// TwinCAT 3 PLC project PLC_v01
// ProgramVersion: 3.1.4022.1
// libraries:
//   Tc2_Math, * (Beckhoff Automation GmbH)
//   Tc2_MC2, * (Beckhoff Automation GmbH)
//   Tc2_MC2_Drive, * (Beckhoff Automation GmbH)
//   Tc2_NCI, * (Beckhoff Automation GmbH)
//   Tc2_NcKinematicTransformation, * (Beckhoff Automation GmbH)
//   Tc2_Standard, * (Beckhoff Automation GmbH)
//   Tc2_System, * (Beckhoff Automation GmbH)
//   Tc2_Utilities, * (Beckhoff Automation GmbH)
//   Tc3_Module, * (Beckhoff Automation GmbH)
//   Tc3_PLCopen_OpcUa, * (Beckhoff Automation GmbH)
//   VisuDialogs, * (System)
// project tree:
//   DUTs/ E_NciChannelState.TcDUT, ST_AxisInterface.TcDUT, ST_AxisInterfaceIn.TcDUT, ST_AxisInterfaceOut.TcDUT, ST_FileDialogParams.TcDUT, ST_OpcUAVariablesR.TcDUT, ST_OpcUAVariablesW.TcDUT (not stored)
//   GVLs/ GVL_Axis.TcGVL, GVL_FileOpen.TcGVL (not stored), GVL_Kin.TcGVL, GVL_Nci.TcGVL, GVL_Process.TcGVL (not stored), GVL_Process_Deneme.TcGVL
//   / PlcTask.TcTTO, Visualization Manager.TcVMO (not stored)
//   POUs/Deneme/ POU_Process_Deneme.TcPOU, POU_VisButton.TcPOU
//   POUs/ FB_AxisControl.TcPOU (not stored), MAIN.TcPOU, PRG_MFuncControl.TcPOU (not stored), PRG_NcControl.TcPOU, PRG_Process.TcPOU (not stored)
//   POUs/KIN/ PRG_Kinematic.TcPOU
//   POUs/NCI/ FB_NciChannel.TcPOU (not stored), FB_NciFastMFunctions.TcPOU, FB_NciMFunctions.TcPOU (not stored), FB_NciReadLine.TcPOU (not stored), FB_NciWriteToolParams.TcPOU (not stored)
//   POUs/OPC-UA/ FB_OpcUAWrite.TcPOU (not stored), PRG_OpcUA.TcPOU (not stored)
//   POUs/UTIL/ FB_Flash.TcPOU (not stored), FB_ScreenOnOff_Win7.TcPOU
//   VISUs/AxisList/ VisuAxisM1.TcVIS, VisuAxisM2.TcVIS, VisuAxisM3.TcVIS, VisuAxisX.TcVIS (not stored), VisuAxisX_1.TcVIS, VisuAxisY.TcVIS, VisuAxisY_1.TcVIS, VisuAxisZ.TcVIS (not stored), VisuAxisZ_1.TcVIS (not stored)
//   VISUs/Frame/ Visualization_FileList.TcVIS, VisuAxisControl.TcVIS, VisuAxisControl_1.TcVIS, VisuAxisInfo.TcVIS (not stored)
//   VISUs/ GlobalTextList.TcGTLO, ImagePool.TcIPO (not stored), Visualization.TcVIS (not stored), Visualization_1.TcVIS, Visualization_AxesInfo.TcVIS, Visualization_AxesInfo_Manual.TcVIS
// real-time tasks:
//   TASK PlcTask: cycle T#10ms, priority 20, ADS port 350
// motion (NC):
//   TASK NC-Task 1 SAF: cycle T#2ms, priority 4, ADS port 501
//   TASK NC-Task 1 SVB: cycle T#10ms, priority 8, ADS port 511
//   AXIS M1 (id 1)
//     Dynamic: Acceleration=120.484, Deceleration=120.484, Jerk=361.452, DelayTime=0.008
//     Velo: RefSearch=0.803225806425292, RefSync=0.803225806425292, SlowManual=10, FastManual=25, Fast=80.3225806425291, Maximum=80.3226
//     OtherSettings: AllowMotionCmdToSlave=true
//     encoder EncType=1
//       EncPara: ScaleFactorNumerator=11.6129032254259, ScaleFactorDenominator=1048576, Offset=-0.7867, Inverse=true
//     drive DrvType=5
//       DrvPara: Inverse=true
//         Analog: VeloReferenz=88.3548387067821, TorqueScale=10, ScaleFactorActTorque=0.1
//         TimeComp: TaskDelayCycles=1
//     controller CtrType=1
//       CtrPara: PriorControlFactor=1
//         PID: PosKp=10
//         Observer: BandWidth=20
//   AXIS M2 (id 2)
//     Dynamic: Acceleration=120.483870963794, Deceleration=120.483870963794, Jerk=361.451612891381, DelayTime=0.008
//     Velo: RefSearch=0.803225806425292, RefSync=0.803225806425292, SlowManual=10, FastManual=25, Fast=80.3225806425291, Maximum=80.3225806425291
//     OtherSettings: AllowMotionCmdToSlave=true
//     encoder EncType=1
//       EncPara: ScaleFactorNumerator=11.6129032254259, ScaleFactorDenominator=1048576, Offset=-4.6881, Inverse=true
//     drive DrvType=5
//       DrvPara: Inverse=true
//         Analog: VeloReferenz=88.3548387067821, TorqueScale=10, ScaleFactorActTorque=0.1
//         TimeComp: TaskDelayCycles=1
//     controller CtrType=1
//       CtrPara: PriorControlFactor=1
//         PID: PosKp=10
//         Observer: BandWidth=20
//   AXIS M3 (id 3)
//     Dynamic: Acceleration=120.483870963794, Deceleration=120.483870963794, Jerk=361.451612891381, DelayTime=0.008
//     Velo: RefSearch=0.803225806425292, RefSync=0.803225806425292, SlowManual=10, FastManual=25, Fast=80.3225806425291, Maximum=80.3225806425291
//     OtherSettings: AllowMotionCmdToSlave=true
//     encoder EncType=1
//       EncPara: ScaleFactorNumerator=11.6129032254259, ScaleFactorDenominator=1048576, Offset=4810.3626, Inverse=true
//     drive DrvType=5
//       DrvPara: Inverse=true
//         Analog: VeloReferenz=88.3548387067821, TorqueScale=10, ScaleFactorActTorque=0.1
//         TimeComp: TaskDelayCycles=1
//     controller CtrType=1
//       CtrPara: PriorControlFactor=1
//         PID: PosKp=10
//         Observer: BandWidth=20
//   AXIS X (id 4)
//     OtherSettings: AllowMotionCmdToSlave=true
//     encoder EncType=1
//     drive DrvType=5
//       Analog: ScaleFactorActTorque=0.1
//       TimeComp: TaskDelayCycles=1
//     controller CtrType=1
//       CtrPara: PriorControlFactor=1
//         Observer: BandWidth=20
//   AXIS Y (id 5)
//     OtherSettings: AllowMotionCmdToSlave=true
//     encoder EncType=1
//     drive DrvType=5
//       Analog: ScaleFactorActTorque=0.1
//       TimeComp: TaskDelayCycles=1
//     controller CtrType=1
//       CtrPara: PriorControlFactor=1
//         Observer: BandWidth=20
//   AXIS Z (id 6)
//     OtherSettings: AllowMotionCmdToSlave=true
//     encoder EncType=1
//     drive DrvType=5
//       Analog: ScaleFactorActTorque=0.1
//       TimeComp: TaskDelayCycles=1
//     controller CtrType=1
//       CtrPara: PriorControlFactor=1
//         Observer: BandWidth=20
// I/O:
//   DEVICE Device 1 (EtherCAT) (disabled), AmsNetId 10.70.16.23.2.1
//     Term 1 (EK1200) [EK1200-5000 EtherCAT Power supply (2A E-Bus)]
//       Term 2 (EL1008) [EL1008 8Ch. Dig. Input 24V, 3ms]
//       Term 3 (EL2008) [EL2008 8Ch. Dig. Output 24V, 0.5A]
//       Term 4 (EL9576) [EL9576 Brake chopper terminal]
//       Term 5 (EL7211-0010) [EL7211-0010 1Ch. MDP742 Servo motor output stage with OCT (50V, 4.5A RMS)]
//       Term 6 (EL7211-0010) [EL7211-0010 1Ch. MDP742 Servo motor output stage with OCT (50V, 4.5A RMS)]
//       Term 7 (EL7211-0010) [EL7211-0010 1Ch. MDP742 Servo motor output stage with OCT (50V, 4.5A RMS)]
//       Term 8 (EL9011) [EL9011 End Terminal]
// variable links:
//   PLC_v01/PLC_v01 Instance <-> NC-Task 1 SAF/Axes/M1
//     PlcTask Inputs/GVL_Axis.AxisM1_B.NcToPlc <-> Outputs/ToPlc
//     PlcTask Outputs/GVL_Axis.AxisM1_B.PlcToNc <-> Inputs/FromPlc
//   PLC_v01/PLC_v01 Instance <-> NC-Task 1 SAF/Axes/M2
//     PlcTask Inputs/GVL_Axis.AxisM2_C.NcToPlc <-> Outputs/ToPlc
//     PlcTask Outputs/GVL_Axis.AxisM2_C.PlcToNc <-> Inputs/FromPlc
//   PLC_v01/PLC_v01 Instance <-> NC-Task 1 SAF/Axes/M3
//     PlcTask Inputs/GVL_Axis.AxisM3_A.NcToPlc <-> Outputs/ToPlc
//     PlcTask Outputs/GVL_Axis.AxisM3_A.PlcToNc <-> Inputs/FromPlc
//   PLC_v01/PLC_v01 Instance <-> NC-Task 1 SAF/Axes/X
//     PlcTask Inputs/GVL_Axis.AxisX.NcToPlc <-> Outputs/ToPlc
//     PlcTask Outputs/GVL_Axis.AxisX.PlcToNc <-> Inputs/FromPlc
//   PLC_v01/PLC_v01 Instance <-> NC-Task 1 SAF/Axes/Y
//     PlcTask Inputs/GVL_Axis.AxisY.NcToPlc <-> Outputs/ToPlc
//     PlcTask Outputs/GVL_Axis.AxisY.PlcToNc <-> Inputs/FromPlc
//   PLC_v01/PLC_v01 Instance <-> NC-Task 1 SAF/Axes/Z
//     PlcTask Inputs/GVL_Axis.AxisZ.NcToPlc <-> Outputs/ToPlc
//     PlcTask Outputs/GVL_Axis.AxisZ.PlcToNc <-> Inputs/FromPlc
//   PLC_v01/PLC_v01 Instance <-> NC-Task 1 SAF/KIN
//     PlcTask Inputs/GVL_Kin.stKinToPLC <-> Outputs/ToPlc
//     PlcTask Outputs/GVL_Kin.stKinFromPLC <-> Inputs/FromPlc
//   PLC_v01/PLC_v01 Instance <-> NC-Task 1 SAF/NCI
//     PlcTask Inputs/GVL_Nci.stNciToPLC <-> Outputs/ToPlc
//     PlcTask Outputs/GVL_Nci.stPlcToNci <-> Inputs/FromPlc

CONFIGURATION PLC_v01
    RESOURCE PLC ON TwinCAT3
        TASK PlcTask(INTERVAL := T#10ms, PRIORITY := 20);
        PROGRAM MAIN WITH PlcTask : MAIN;
    END_RESOURCE
END_CONFIGURATION

// ---- DUTs/E_NciChannelState.TcDUT
TYPE E_NciChannelState :
(
	eNCI_INTERPRETER_INITFAILED := 0, 
	eNCI_INTERPRETER_IDLE := 1, 
	eNCI_INTERPRETER_READY := 2,
	eNCI_INTERPRETER_STARTED := 3, 
	eNCI_INTERPRETER_SCANNING := 4, 
	eNCI_INTERPRETER_RUNNING := 5,
	eNCI_INTERPRETER_STAY_RUNNING := 6,
	eNCI_INTERPRETER_WRITETABLE := 7,
	eNCI_INTERPRETER_SEARCHLINE := 8, 
	eNCI_INTERPRETER_END := 9,
	eNCI_INTERPRETER_SINGLESTOP := 10,
	eNCI_INTERPRETER_ABORTING := 11,
	eNCI_INTERPRETER_ABORTED := 12, 
	eNCI_INTERPRETER_FAULT := 13,
	eNCI_INTERPRETER_RESET := 14, 
	eNCI_INTERPRETER_STOP := 15,
	eNCI_INTERPRETER_WAITFUNC := 16,
	eNCI_INTERPRETER_FLUSHBUFFERS := 17
);
END_TYPE

// ---- DUTs/ST_AxisInterface.TcDUT
TYPE ST_AxisInterface :
STRUCT
	In		: ST_AxisInterfaceIn;
	Out		: ST_AxisInterfaceOut;
END_STRUCT
END_TYPE

// ---- DUTs/ST_AxisInterfaceIn.TcDUT
TYPE ST_AxisInterfaceIn :
STRUCT
	xEnable			: BOOL;
	xReset			: BOOL;
	xDriveReset		: BOOL;
	xMove			: BOOL;
	xHome			: BOOL;
	xHomeSensor		: BOOL;
	xJogFw			: BOOL;
	xJogBw			: BOOL;
	fHomePos		: LREAL;
	fSetPos			: LREAL;
	fSetVelo		: LREAL;
	fSetAcc			: LREAL;
	fSetDec			: LREAL;
	fSetJerk		: LREAL;
	fJogVelo		: LREAL	:= 20;
	fOverride		: LREAL	:= 100.0;
END_STRUCT
END_TYPE

// ---- DUTs/ST_AxisInterfaceOut.TcDUT
TYPE ST_AxisInterfaceOut :
STRUCT
	xEnabled		: BOOL;
	xHomed			: BOOL;
	xMoveDone		: BOOL;
	xAxisError		: BOOL;
	nAxisErrId		: UDINT;
	xDriveError		: BOOL;
	nDriveErrId		: UDINT;
	xFunctionError	: BOOL;
	nFunctionErrId	: UDINT;
END_STRUCT
END_TYPE

// ---- DUTs/ST_FileDialogParams.TcDUT
TYPE ST_FileDialogParams :
STRUCT
	sTitle 		: STRING;
	sDirectory 	: STRING(255);
	sFile 		: STRING(255);
	sFilter 	: STRING;
	bInit 		: BOOL;
END_STRUCT
END_TYPE

// ---- DUTs/ST_OpcUAVariablesR.TcDUT
TYPE ST_OpcUAVariablesR :
STRUCT
	bEnableAllProcess	: BOOL;
	bNciStart			: BOOL;
END_STRUCT
END_TYPE

// ---- GVLs/GVL_Axis.TcGVL
VAR_GLOBAL
// Kullanilacak olan gercek eksenler
	AxisM1_B			: AXIS_REF;			
	AxisM2_C			: AXIS_REF;
	AxisM3_A			: AXIS_REF;	
	
// Kinematik grupta olusacak eksenler
	AxisX				: AXIS_REF;
	AxisY				: AXIS_REF;
	AxisZ				: AXIS_REF;
	
// Gercek eksenler icin interface yapilari
	stAxisM1_B			: ST_AxisInterface;
	stAxisM2_C			: ST_AxisInterface;
	stAxisM3_A			: ST_AxisInterface;
	
// Kinematik eksenlerin interface yapilari
	stAxisX				: ST_AxisInterface;
	stAxisY				: ST_AxisInterface;
	stAxisZ				: ST_AxisInterface;
	
	sAxisM1_BName		: STRING	:= 'Axis M1';
	sAxisM2_CName		: STRING	:= 'Axis M2';
	sAxisM3_AName		: STRING	:= 'Axis M3';
	
	
	sAxisXName			: STRING	:= 'Axis X';
	sAxisYName			: STRING	:= 'Axis Y';
	sAxisZName			: STRING	:= 'Axis Z';
	
	AxisM1PosValue		: LREAL;
	AxisM2PosValue		: LREAL;
	AxisM3PosValue		: LREAL;
	
	AxisXVal	:	LREAL;
	AxisYVal	:	LREAL;	
	AxisZVal	:	LREAL;
	
END_VAR

// ---- GVLs/GVL_Kin.TcGVL
{attribute 'qualified_only'}
VAR_GLOBAL
	stKinToPLC			AT%I*	: NCTOPLC_NCICHANNEL_REF;
	stKinFromPLC		AT%Q*	: PLCTONC_NCICHANNEL_REF;
	
	stAxesList					: ST_KinAxes;
	
END_VAR

// ---- GVLs/GVL_Nci.TcGVL
VAR_GLOBAL
	stNciToPLC	AT%I*		: NCTOPLC_NCICHANNEL_REF;
	stPlcToNci	AT%Q*		: PLCTONC_NCICHANNEL_REF;
	
	bMFunc					: ARRAY[0..cnMaxMFuncNumber] OF BOOL;
	bQuitMFunc				: ARRAY[0..cnMaxMFuncNumber] OF BOOL;
	bFastMFunc				: ARRAY[0..cnMaxMFuncNumber] OF BOOL;
	
	fNciRParamsWrite		: ARRAY[cnStartIndexWriteRParam..cnEndIndexWriteRParam] OF LREAL;
	fNciRParamsRead			: ARRAY[cnStartIndexReadRParam..cnEndIndexReadRParam] OF LREAL;
	stNciToolParams			: ARRAY[1..cnMaxToolNumber] OF ToolDesc;
END_VAR
VAR_GLOBAL CONSTANT
	cnMaxMFuncNumber		: INT	:= 159;
	cnStartIndexWriteRParam	: INT	:= 0;
	cnEndIndexWriteRParam	: INT	:= 100;
	cnStartIndexReadRParam	: INT	:= 101;
	cnEndIndexReadRParam	: INT	:= 201;
	cnMaxToolNumber			: INT	:= 10;
END_VAR

// ---- GVLs/GVL_Process_Deneme.TcGVL
{attribute 'qualified_only'}
VAR_GLOBAL
	
bSensor	:	BOOL;
bCatch	:	BOOL;

bMovementDone	:	BOOL;
bDataComp	:	BOOL;
bGrapDone	:	BOOL;
END_VAR

// ---- POUs/MAIN.TcPOU
PROGRAM MAIN
VAR
	sFilePathName	: STRING := 'C:\TwinCAT\CNC\TestNci1.txt';
	sErrorMessage	: STRING := '';
	bOpen			: BOOL;
	bClose 			: BOOL;
	bSave 			: BOOL;
	bNew			: BOOL;
	nErrorCode		: USINT;
	nLineNumber		: USINT;
	bEnable: BOOL;
END_VAR



sErrorMessage	:= VisuFctTextEditorGetErrorText(usiErrCode := nErrorCode);

PRG_NcControl();
//PRG_MFuncControl();
PRG_Kinematic();

//PRG_Process();

//PRG_OpcUA();

//POU_VisButton();
POU_Process_Deneme();


	PRG_Kinematic.bExecuteKinConfigGroup;
	
	
	stAxisX.In.fSetPos;
	stAxisY.In.fSetPos;
	stAxisZ.In.fSetPos;

	
	stAxisX.In.xMove;
	stAxisY.In.xMove;
	stAxisZ.In.xMove;



AxisM1PosValue	:=	LMOD(AxisM1_B.NcToPlc.ModuloActPos,360);
AxisM2PosValue	:=	LMOD(AxisM2_C.NcToPlc.ModuloActPos,360);
AxisM3PosValue	:=	LMOD(AxisM3_A.NcToPlc.ModuloActPos,360);



	
	
	AxisXVal	:=	AxisX.NcToPlc.ActPos;
	AxisYVal	:=	AxisY.NcToPlc.ActPos;
	AxisZVal	:=	AxisZ.NcToPlc.ActPos;

END_PROGRAM

// ---- POUs/PRG_NcControl.TcPOU
PROGRAM PRG_NcControl
VAR_INPUT
	//PRG_Process içerisinde resetlemede kullanabilmek için 
	bNciEnable			: BOOL;
	bNciStart			: BOOL;
END_VAR

VAR
	fbAxisControlM1_B	: FB_AxisControl;
	fbAxisControlM2_C	: FB_AxisControl;
	fbAxisControlM3_A	: FB_AxisControl;	
	
	fbAxisControlX		: FB_AxisControl;
	fbAxisControlY		: FB_AxisControl;
	fbAxisControlZ		: FB_AxisControl;
	
	fbNciChannel		: FB_NciChannel;
	fbNciMFunc			: FB_NciMFunctions;
	fbNciFastMFunc		: FB_NciFastMFunctions;
	fbNciReadLine		: FB_NciReadLine;
	bAxisEnable			: BOOL;
	fAxisOverride		: LREAL;
	bNciSingleMode		: BOOL;
	bNciNextStep		: BOOL;
	fNciOverride		: LREAL	:= 100.0;
	eNciItpState		: E_NciChannelState;
	bBuildGroupDone		: BOOL;
	bSingleModeActive	: BOOL;
	bProgramRunning		: BOOL;
	bProgramStopped		: BOOL;
	bProgramFinished	: BOOL;
	bNciError			: BOOL;
	nNciErrorId			: UDINT;
	bMFuncBusy			: BOOL;
	bMFuncError			: BOOL;
	nMFuncErrorId		: UDINT;
	bEnableReadLine		: BOOL	:= TRUE;
	sNciLines			: STRING(255);
	sNciActualLine		: STRING(80);	
	bEnable: BOOL;
END_VAR

//ACT_EmergencyOnPanel();

fbAxisControlM1_B(stAxisInterface:= stAxisM1_B, stAxisRef:= AxisM1_B);
fbAxisControlM2_C(stAxisInterface:= stAxisM2_C, stAxisRef:= AxisM2_C);
fbAxisControlM3_A(stAxisInterface:= stAxisM3_A, stAxisRef:= AxisM3_A);

fbAxisControlX(stAxisInterface:= stAxisX, stAxisRef:= AxisX);
fbAxisControlY(stAxisInterface:= stAxisY, stAxisRef:= AxisY);
fbAxisControlZ(stAxisInterface:= stAxisZ, stAxisRef:= AxisZ);

(*
		stAxisX.In.xEnable		:= bEnable;
		stAxisY.In.xEnable		:= bEnable;
		stAxisZ.In.xEnable		:= bEnable;
		stAxisM1_B.In.xEnable	:= bEnable;
		stAxisM2_C.In.xEnable	:= bEnable;
		stAxisM3_A.In.xEnable	:= bEnable;
*)
(*		
fbNciChannel(
	bEnable				:= bNciEnable, 
	bStart				:= bNciStart, 
	bSingleMode			:= bNciSingleMode,
	bSingleModeStart	:= bNciNextStep,
	fOverride			:= fNciOverride,
	nXAxisId			:= AxisX.NcToPlc.AxisId, 
	nYAxisId			:= AxisY.NcToPlc.AxisId, 
	nZAxisId			:= AxisZ.NcToPlc.AxisId, 
	sProgramPath		:= PRG_Process.sFileName, 
	sSubroutinePath		:= 'C:\TwinCAT\Mc\Nci\Sub\', 
	sNciToPLC			:= stNciToPLC, 
	sPlcToNci			:= stPlcToNci, 
	eNciChannelState	=> eNciItpState, 
	bBuildGroupDone		=> bBuildGroupDone, 
	bSingleModeActive	=> bSingleModeActive,
	bProgramRunning		=> bProgramRunning, 
	bProgramStopped		=> bProgramStopped, 
	bProgramFinished	=> bProgramFinished, 
	bError				=> bNciError, 
	nErrorId			=> nNciErrorId);
	
fbNciMFunc(
	sNciToPlc			:= stNciToPLC, 
	sPlcToNci			:= stPlcToNci, 
	bBusy				=> bMFuncBusy, 
	bError				=> bMFuncError, 
	nErrorId			=> nMFuncErrorId);
	
fbNciFastMFunc(
	sNciToPlc			:= stNciToPLC);
	
fbNciReadLine(
	bEnable				:= bEnableReadLine, 
	tIdleTime			:= T#100MS, 
	sNciToPlc			:= stNciToPLC, 
	sNciLines			=> sNciLines,
	sActualLine			=> sNciActualLine );
	

*)

ACTION ACT_EmergencyOnPanel:
(*Button On Control Panel- Emergency and Green Button*)
GVL_Process.fTrigbEmergency(CLK:= GVL_Process.bEmergencyOnPanel);
GVL_Process.rTrigbEmergency(CLK:= GVL_Process.bEmergencyOnPanel);


CASE GVL_Process.nStateEmergency OF 
0:
	IF GVL_Process.fTrigbEmergency.Q THEN 
		fNciOverride	:= 0;
		GVL_Process.nStateEmergency	:= 10;
	END_IF
	
10:
	IF GVL_Process.rTrigbEmergency.Q THEN 
		GVL_Process.nStateEmergency	:= 20;
	END_IF
	
20:
	IF GVL_Process.bGreenBtnOnPanel THEN 
		fNciOverride	:= 100;
		GVL_Process.nStateEmergency	:= 0;
	END_IF
END_CASE
END_ACTION

END_PROGRAM

// ---- POUs/NCI/FB_NciFastMFunctions.TcPOU
FUNCTION_BLOCK FB_NciFastMFunctions
VAR_IN_OUT
	sNciToPlc		: NCTOPLC_NCICHANNEL_REF;
END_VAR
VAR_OUTPUT
END_VAR
VAR
	i				: INT;
	l				: SINT;
	bBit			: BOOL;
	index			: UINT;
END_VAR


(* Fill the global defined M-functions array with 
	fast M-Functions from NCI Channel *)

FOR i:=0 TO 4 DO  (* check all 5 dwords *)
	FOR l := 0 TO 31 DO
		bBit := GETBIT32(sNciToPlc.FastMFuncMask[i+1], l);
      	index := INT_TO_UINT((i*32) + l);
		IF ( bBit ) THEN
			bFastMFunc[index] := TRUE;
		ELSE
			bFastMFunc[index] := FALSE;
		END_IF
	END_FOR
END_FOR

END_FUNCTION_BLOCK

// ---- POUs/KIN/PRG_Kinematic.TcPOU
PROGRAM PRG_Kinematic
VAR_INPUT
		bExecuteKinConfigGroup	: BOOL;
		bCartesianMode			: BOOL := TRUE;
		bExecuteKinResetGroup	: BOOL;
END_VAR
VAR
	fbKinConfigGroup			: FB_KinConfigGroup;
	fbKinResetGroup				: FB_KinResetGroup;
	eKinStatus					: E_KinStatus;
END_VAR


GVL_Kin.stAxesList.nAxisIdsAcs[1]	:= AxisM1_B.NcToPlc.AxisId;
GVL_Kin.stAxesList.nAxisIdsAcs[2]	:= AxisM2_C.NcToPlc.AxisId;
GVL_Kin.stAxesList.nAxisIdsAcs[3]	:= AxisM3_A.NcToPlc.AxisId;

GVL_Kin.stAxesList.nAxisIdsMcs[1]	:= AxisX.NcToPlc.AxisId;
GVL_Kin.stAxesList.nAxisIdsMcs[2]	:= AxisY.NcToPlc.AxisId;
GVL_Kin.stAxesList.nAxisIdsMcs[3]	:= AxisZ.NcToPlc.AxisId;

ItpSetOverridePercent(100.0, GVL_Kin.stKinFromPLC);

fbKinConfigGroup(
	bExecute		:= bExecuteKinConfigGroup, 
	bCartesianMode	:= bCartesianMode, 
	stAxesList		:= GVL_Kin.stAxesList, 
	stKinRefIn		:= GVL_Kin.stKinToPLC);	
	
fbKinResetGroup(
	bExecute		:= bExecuteKinResetGroup, 
	nItpChannelId	:= ItpGetChannelId(GVL_Kin.stKinToPLC), 
	stKinRefIn		:= GVL_Kin.stKinToPLC, 
	stAxesList		:= GVL_Kin.stAxesList);

END_PROGRAM

// ---- POUs/Deneme/POU_Process_Deneme.TcPOU
PROGRAM POU_Process_Deneme
VAR
	nStateProcess: INT;
	bSystemStart: BOOL;
	bSensor: BOOL;
	T1: TON;
	T2: TON;
	rtrig_Obj: R_TRIG;
END_VAR

		
	stAxisM1_B.In.xEnable	:= TRUE;
	stAxisM2_C.In.xEnable	:= TRUE;
	stAxisM3_A.In.xEnable	:= TRUE;
	
	stAxisX.In.xEnable	:= TRUE;
	stAxisY.In.xEnable	:= TRUE;
	stAxisZ.In.xEnable	:= TRUE;
		
	stAxisM1_B.In.fOverride	:= 100;
	stAxisM2_C.In.fOverride	:= 100;
	stAxisM3_A.In.fOverride	:= 100;
	
	stAxisX.In.fOverride	:= 100;
	stAxisY.In.fOverride	:= 100;
	stAxisZ.In.fOverride	:= 100;
	

	
CASE nStateProcess	OF
	
0:
IF bSystemStart THEN


	PRG_Kinematic.bExecuteKinConfigGroup	:=	TRUE;
	stAxisX.In.xMove	:=	TRUE;
	stAxisY.In.xMove	:=	TRUE;
	stAxisZ.In.xMove	:=	TRUE;

			
	stAxisX.In.fSetVelo	:=50;
	stAxisY.In.fSetVelo	:=50;
	stAxisZ.In.fSetVelo	:=50;

	IF 
	PRG_Kinematic.fbKinConfigGroup.bDone AND 
	stAxisX.Out.xEnabled	AND
	stAxisY.Out.xEnabled	AND
	stAxisZ.Out.xEnabled	THEN
	
	

		nStateProcess	:=	10;
	
	ELSIF	PRG_Kinematic.fbKinConfigGroup.bError THEN
		nStateProcess	:=	1000;
	END_IF	
	
END_IF

10:
GVL_Process_Deneme.bMovementDone	:=	FALSE;
GVL_Process_Deneme.bDataComp	:=FALSE;


IF	GVL_Process_Deneme.bSensor	THEN
	
	GVL_Process_Deneme.bMovementDone	:=	TRUE;
	
	stAxisX.In.fSetPos	:=	0;
	stAxisY.In.fSetPos	:=	0;
	stAxisZ.In.fSetPos	:=	-400;
	

	IF 	stAxisX.Out.xMoveDone	AND stAxisY.Out.xMoveDone	AND stAxisZ.Out.xMoveDone THEN 
	
	GVL_Process_Deneme.bCatch	:=	TRUE;
	
	GVL_Process_Deneme.bMovementDone	:=	FALSE;				//Malzeme Alındı


	
	nStateProcess	:=	20;
	
	ELSIF stAxisX.Out.xAxisError	OR
	stAxisY.Out.xAxisError	OR
	stAxisZ.Out.xAxisError	OR
	stAxisM1_B.Out.xAxisError	OR
	stAxisM2_C.Out.xAxisError	OR	
	stAxisM3_A.Out.xAxisError	THEN

	nStateProcess	:=	999;	
	
END_IF
	
	
	
END_IF

20:

stAxisX.In.fSetVelo	:=300;
stAxisY.In.fSetVelo	:=300;
stAxisZ.In.fSetVelo	:=300;


stAxisZ.In.fSetPos	:=	-370;			//Alınan malzeme bırakılacağı konuma götürüldü
stAxisY.In.fSetPos	:=	310;

nStateProcess	:=	25;


25:

	IF  stAxisY.Out.xMoveDone	AND stAxisZ.Out.xMoveDone THEN 

	
	nStateProcess	:=	30;
	
	ELSIF stAxisX.Out.xAxisError	OR
	stAxisY.Out.xAxisError	OR
	stAxisZ.Out.xAxisError	OR
	stAxisM1_B.Out.xAxisError	OR
	stAxisM2_C.Out.xAxisError	OR	
	stAxisM3_A.Out.xAxisError	THEN

	nStateProcess	:=	999;	
	
END_IF
	
30:
stAxisX.In.fSetVelo	:=50;
stAxisY.In.fSetVelo	:=50;
stAxisZ.In.fSetVelo	:=50;

stAxisZ.In.fSetPos	:=	-400;		



	IF stAxisZ.Out.xMoveDone THEN 

	GVL_Process_Deneme.bDataComp	:=	TRUE;	// Malzeme bırakıldı
	
//	GVL_Process_Deneme.bMovementDone	:=	TRUE;

	GVL_Process_Deneme.bCatch	:=	FALSE;
	
	
	nStateProcess	:=	40;
	
	
	ELSIF stAxisX.Out.xAxisError	OR
	stAxisY.Out.xAxisError	OR
	stAxisZ.Out.xAxisError	OR
	stAxisM1_B.Out.xAxisError	OR
	stAxisM2_C.Out.xAxisError	OR	
	stAxisM3_A.Out.xAxisError	THEN

	nStateProcess	:=	999;	
	
END_IF


40:

stAxisX.In.fSetVelo	:=1000;
stAxisY.In.fSetVelo	:=1000;
stAxisZ.In.fSetVelo	:=1000;


stAxisX.In.fSetPos	:=	0;
stAxisY.In.fSetPos	:=	0;
stAxisZ.In.fSetPos	:=	-370;

nStateProcess	:=	45;

45:
		
	IF 	stAxisX.Out.xMoveDone	AND stAxisY.Out.xMoveDone	 THEN 


	GVL_Process_Deneme.bDataComp	:=FALSE;
		GVL_Process_Deneme.bMovementDone	:=FALSE;

	
	nStateProcess	:=	0;
	
	
	ELSIF stAxisX.Out.xAxisError	OR
	stAxisY.Out.xAxisError	OR
	stAxisZ.Out.xAxisError	OR
	stAxisM1_B.Out.xAxisError	OR
	stAxisM2_C.Out.xAxisError	OR	
	stAxisM3_A.Out.xAxisError	THEN

	nStateProcess	:=	999;	
	
END_IF





END_CASE

END_PROGRAM

// ---- POUs/Deneme/POU_VisButton.TcPOU
PROGRAM POU_VisButton
VAR
	
xUp	:	BOOL;
xDown	:	BOOL;

yUp	:	BOOL;
yDown	:	BOOL;

zuP	:	BOOL;	
zDown	:	BOOL;

DecVal	:	LREAL;



	xUpR_TRIG: R_TRIG;
	xDownR_TRIG: R_TRIG;
	yUpR_TRIG: R_TRIG;
	yDownR_TRIG: R_TRIG;
	zUpR_TRIG: R_TRIG;
	zDownR_TRIG: R_TRIG;
	BridgeValZ: LREAL;
END_VAR

	
xUpR_TRIG(CLK:=xUp , Q=> );
xDownR_TRIG(CLK:=xDown , Q=> );

yUpR_TRIG(CLK:=yUp , Q=> );
yDownR_TRIG(CLK:=yDown , Q=> );

zUpR_TRIG(CLK:=zUp , Q=> );
zDownR_TRIG(CLK:=zDown , Q=> );


stAxisZ.In.fSetPos	:=	BridgeValZ;

	//stAxisX.In.fSetPos;
	//stAxisY.In.fSetPos;
	//stAxisZ.In.fSetPos;

IF xUpR_TRIG.Q	THEN
	
stAxisX.In.fSetPos	:=	stAxisX.In.fSetPos	+	10;


ELSIF xDownR_TRIG.Q THEN
	stAxisX.In.fSetPos	:=	stAxisX.In.fSetPos	-	10;
END_IF



IF yUpR_TRIG.Q	THEN
	
stAxisY.In.fSetPos	:=	stAxisY.In.fSetPos	+	10;


ELSIF yDownR_TRIG.Q THEN
	stAxisY.In.fSetPos	:=	stAxisY.In.fSetPos	-	10;
END_IF




IF zUpR_TRIG.Q	THEN
	
BridgeValZ	:=	BridgeValZ	+	10;


ELSIF zDownR_TRIG.Q THEN
	BridgeValZ	:=	BridgeValZ	-	10;
END_IF

END_PROGRAM

// ---- POUs/UTIL/FB_ScreenOnOff_Win7.TcPOU
FUNCTION_BLOCK FB_ScreenOnOff_Win7
VAR_INPUT
	bScreenOff			: BOOL;
END_VAR
VAR_OUTPUT
	bDone				: BOOL;
END_VAR
VAR
	fbSleepMonitor		: NT_StartProcess;
	nState				: INT;
END_VAR

CASE nState OF 	
0:
	IF bScreenOff THEN
		nState	:= 10;
	END_IF
	
10:
	fbSleepMonitor(
		NETID		:= '', 
		PATHSTR		:= 'C:\MonitorSleep.exe', 
		DIRNAME		:= 'C:\', 
		COMNDLINE	:= , 
		START		:= TRUE, 
		TMOUT		:= T#5S, 
		BUSY		=> , 
		ERR			=> , 
		ERRID		=> );
	
	IF NOT fbSleepMonitor.BUSY AND NOT fbSleepMonitor.ERR THEN 
		fbSleepMonitor(START := FALSE);
		nState		:= 20;
	END_IF 
		
20:
	bDone	:= TRUE;
	IF NOT bScreenOff THEN 
		bDone 	:= FALSE;
		nState	:= 0;
	END_IF 		

END_CASE

END_FUNCTION_BLOCK

// ---- VISUs/AxisList/VisuAxisM1.TcVIS
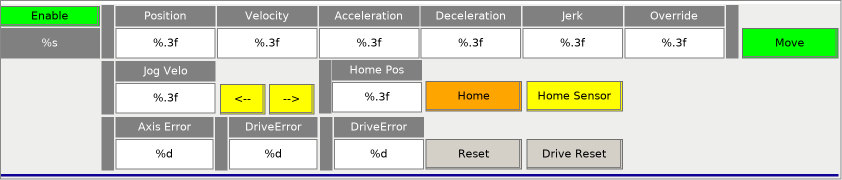
VISUALIZATION VisuAxisM1  // 842x180
    Frame (0,4 840x174)
        shows VisuAxisControl(sAxisName := sAxisM1_BName, stAxisVisu := stAxisM1_B)
END_VISUALIZATION

// ---- VISUs/AxisList/VisuAxisM2.TcVIS
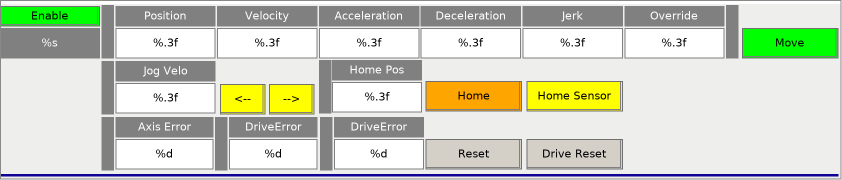
VISUALIZATION VisuAxisM2  // 842x180
    Frame (0,4 840x174)
        shows VisuAxisControl(sAxisName := sAxisM2_CName, stAxisVisu := stAxisM2_C)
END_VISUALIZATION

// ---- VISUs/AxisList/VisuAxisM3.TcVIS
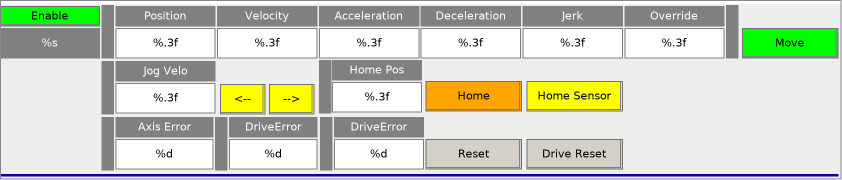
VISUALIZATION VisuAxisM3  // 842x180
    Frame (0,4 840x174)
        shows VisuAxisControl(sAxisName := sAxisM3_AName, stAxisVisu := stAxisM3_A)
END_VISUALIZATION

// ---- VISUs/AxisList/VisuAxisX_1.TcVIS
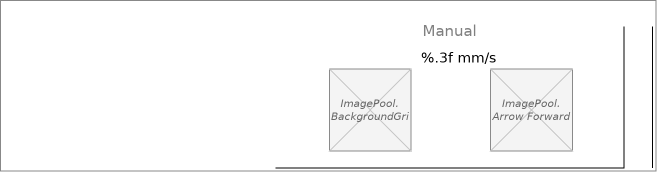
VISUALIZATION VisuAxisX_1  // 657x172
    Frame (0,0 655x170)
        shows VisuAxisControl_1(sAxisName_1 := sAxisXName, stAxisVisu_1 := stAxisX)
END_VISUALIZATION

// ---- VISUs/AxisList/VisuAxisY.TcVIS
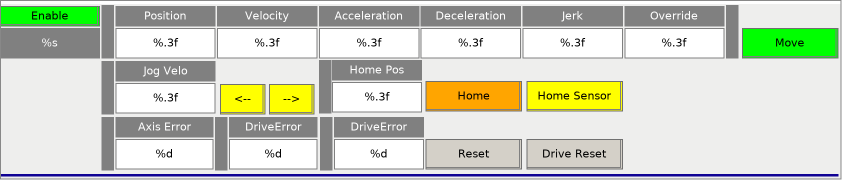
VISUALIZATION VisuAxisY  // 842x180
    Frame (0,4 840x174)
        shows VisuAxisControl(sAxisName := sAxisYName, stAxisVisu := stAxisY)
END_VISUALIZATION

// ---- VISUs/AxisList/VisuAxisY_1.TcVIS
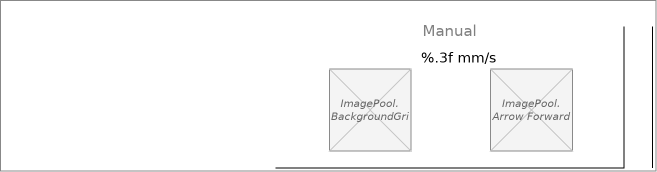
VISUALIZATION VisuAxisY_1  // 657x172
    Frame (0,0 655x170)
        shows VisuAxisControl_1(sAxisName_1 := sAxisYName, stAxisVisu_1 := stAxisY)
END_VISUALIZATION

// ---- VISUs/Frame/Visualization_FileList.TcVIS
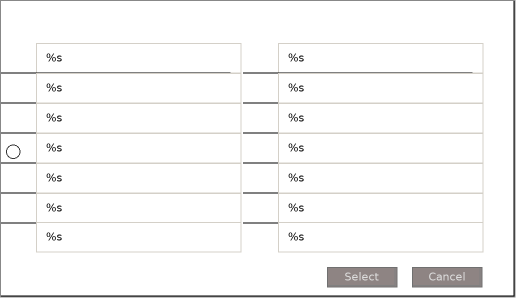
VISUALIZATION Visualization_FileList  // 516x298
    Rectangle (-1,0 515x296)
    Textfield (36,43 205x30), "%s", text variable: PRG_Process.arrFileNameList[1]
    Label (181,-2 158x39), "G-Code List"
    Line (230,73) (1,73)
    Line (230,103) (1,103)
    Line (230,133) (1,133)
    Line (230,163) (1,163)
    Line (230,193) (1,193)
    Line (230,223) (1,223)
    Textfield (36,73 205x30), "%s", text variable: PRG_Process.arrFileNameList[2]
    Textfield (36,103 205x30), "%s", text variable: PRG_Process.arrFileNameList[3]
    Textfield (36,133 205x30), "%s", text variable: PRG_Process.arrFileNameList[4]
    Textfield (36,163 205x30), "%s", text variable: PRG_Process.arrFileNameList[5]
    Textfield (36,193 205x30), "%s", text variable: PRG_Process.arrFileNameList[6]
    Textfield (36,222 205x30), "%s", text variable: PRG_Process.arrFileNameList[7]
    Textfield (278,43 205x30), "%s", text variable: PRG_Process.arrFileNameList[8]
    Line (472,73) (243,73)
    Line (472,103) (243,103)
    Line (472,133) (243,133)
    Line (472,163) (243,163)
    Line (472,193) (243,193)
    Line (472,223) (243,223)
    Textfield (278,73 205x30), "%s", text variable: PRG_Process.arrFileNameList[9]
    Textfield (278,103 205x30), "%s", text variable: PRG_Process.arrFileNameList[10]
    Textfield (278,133 205x30), "%s", text variable: PRG_Process.arrFileNameList[11]
    Textfield (278,163 205x30), "%s", text variable: PRG_Process.arrFileNameList[12]
    Textfield (278,193 205x30), "%s", text variable: PRG_Process.arrFileNameList[13]
    Textfield (278,222 205x30), "%s", text variable: PRG_Process.arrFileNameList[14]
    RadioButton (4,43 488x217), variable: PRG_Process.nFileNameList
    Button (327,267 70x20), "Select"
        tap PRG_Process.bSelectFile
    Button (412,267 70x20), "Cancel"
        tap PRG_Process.bCancelSelectFile
END_VISUALIZATION

// ---- VISUs/Frame/VisuAxisControl.TcVIS
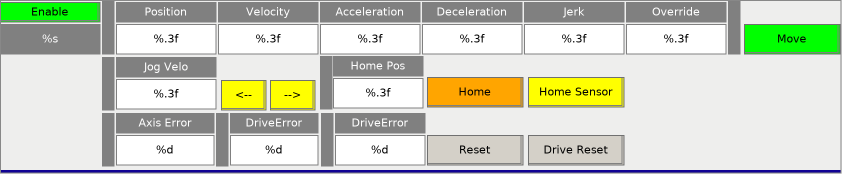
VISUALIZATION VisuAxisControl  // 842x174
VAR_IN_OUT
	sAxisName		: STRING;
	stAxisVisu		: ST_AxisInterface;
END_VAR
    Rectangle (0,24 100x30), "%s", text variable: sAxisName
    Rectangle (116,24 100x30), "%.3f", text variable: stAxisVisu.In.fSetPos
        OnMouseClick: write the text variable via VisuDialogs.Numpad
    Rectangle (116,2 100x20), "Position"
    Rectangle (218,24 100x30), "%.3f", text variable: stAxisVisu.In.fSetVelo
        OnMouseClick: write the text variable via VisuDialogs.Numpad
    Rectangle (218,2 100x20), "Velocity"
    Rectangle (320,24 100x30), "%.3f", text variable: stAxisVisu.In.fSetAcc
        OnMouseClick: write the text variable via VisuDialogs.Numpad
    Rectangle (320,2 100x20), "Acceleration"
    Rectangle (422,24 100x30), "%.3f", text variable: stAxisVisu.In.fSetDec
        OnMouseClick: write the text variable via VisuDialogs.Numpad
    Rectangle (422,2 100x20), "Deceleration"
    Rectangle (524,24 100x30), "%.3f", text variable: stAxisVisu.In.fSetJerk
        OnMouseClick: write the text variable via VisuDialogs.Numpad
    Rectangle (524,2 100x20), "Jerk"
    Rectangle (626,24 100x30), "%.3f", text variable: stAxisVisu.In.fOverride
        OnMouseClick: write the text variable via VisuDialogs.Numpad
    Rectangle (626,2 100x20), "Override"
    Rectangle (116,79 100x30), "%.3f", text variable: stAxisVisu.In.fJogVelo
        OnMouseClick: write the text variable via VisuDialogs.Numpad
    Rectangle (116,57 100x20), "Jog Velo"
    Rectangle (333,78 90x30), "%.3f", text variable: stAxisVisu.In.fHomePos
        OnMouseClick: write the text variable via VisuDialogs.Numpad
    Rectangle (333,56 90x20), "Home Pos"
    Button (0,2 100x20), "Enable"
        toggle stAxisVisu.In.xEnable
    RoundedRectangle (728,1 12x53), colour toggle: stAxisVisu.Out.xMoveDone
    Button (221,80 45x30), "<--"
        tap stAxisVisu.In.xJogBw
    Button (270,80 45x30), "-->"
        tap stAxisVisu.In.xJogFw
    Button (427,77 96x30), "Home"
        toggle stAxisVisu.In.xHome
    Button (528,77 96x30), "Home Sensor"
        toggle stAxisVisu.In.xHomeSensor
    RoundedRectangle (320,56 12x53), colour toggle: stAxisVisu.Out.xHomed
    RoundedRectangle (102,57 12x53)
    RoundedRectangle (102,1 12x53), colour toggle: stAxisVisu.Out.xEnabled
    Button (744,24 96x30), "Move"
        toggle stAxisVisu.In.xMove
    Rectangle (116,135 98x30), "%d", text variable: stAxisVisu.Out.nAxisErrId
    Rectangle (116,113 98x20), "Axis Error"
    RoundedRectangle (102,113 12x53), colour toggle: stAxisVisu.Out.xAxisError
    Rectangle (230,135 88x30), "%d", text variable: stAxisVisu.Out.nDriveErrId
    Rectangle (230,113 88x20), "DriveError"
    RoundedRectangle (216,113 12x53), colour toggle: stAxisVisu.Out.xDriveError
    Rectangle (335,135 90x30), "%d", text variable: stAxisVisu.Out.nFunctionErrId
    Rectangle (335,113 90x20), "DriveError"
    RoundedRectangle (321,113 12x53), colour toggle: stAxisVisu.Out.xFunctionError
    Button (427,135 96x30), "Reset"
        tap stAxisVisu.In.xReset
    Button (528,135 96x30), "Drive Reset"
        tap stAxisVisu.In.xDriveReset
    RoundedRectangle (0,170 840x2)
END_VISUALIZATION

// ---- VISUs/Frame/VisuAxisControl_1.TcVIS
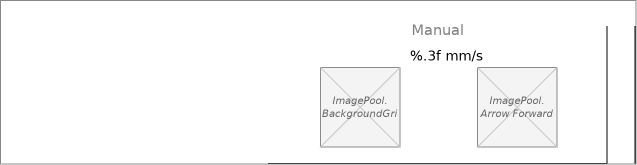
VISUALIZATION VisuAxisControl_1  // 637x165, background image ImagePool.BackgrounFrame
VAR_IN_OUT
	sAxisName_1		: STRING;
	stAxisVisu_1	: ST_AxisInterface;
END_VAR
    Line (635,163) (635,26), invisible if: PRG_Process.bInvisible
    Ellipse (333,77 52x55), invisible if: not stAxisVisu_1.In.xJogBw
    Image (320,67 80x80), image: ImagePool.BackgroundGri
    Ellipse (490,78 52x55), invisible if: not stAxisVisu_1.In.xJogFw
    Image (477,67 80x80), image: ImagePool.Arrow Forward
    Label (374,10 132x40), "Manual"
    Rectangle (389,42 97x28), "%.3f mm/s", text variable: stAxisVisu_1.In.fJogVelo
        OnMouseClick: write the text variable via VisuDialogs.Numpad
    Line (268,163) (607,163)
    InvisibleInput (323,67 86x78)
        tap stAxisVisu_1.In.xJogBw
    InvisibleInput (478,68 81x76)
        tap stAxisVisu_1.In.xJogFw
    Line (607,163) (607,26)
END_VISUALIZATION

// ---- VISUs/GlobalTextList.TcGTLO
TEXTLIST GlobalTextList
  116 = ''
  114 = '           %s'
  113 = '      %s'
  115 = '  %s'
  37 = ' %s'
  74 = ' M1'
  76 = ' M3'
  77 = ' X'
  78 = ' Y'
  79 = ' Z'
  204 = '%'
  11 = '%.1f'
  8 = '%.2f'
  1 = '%.3f'
  96 = '%.3f mm/s'
  1129 = '%.4f'
  68 = '%a'
  13 = '%d'
  845 = '%f'
  494 = '%i'
  19 = '%s'
  69 = '%t %a'
  28 = '-->'
  27 = '<--'
  20 = 'Acceleration'
  117 = 'ACS'
  4 = 'Act. Position'
  9 = 'Act. Velocity'
  100 = 'AUTOMATIC MODE'
  18 = 'Axis'
  72 = 'Axis Coordinate System'
  32 = 'Axis Error'
  6 = 'Axis List'
  94 = 'Axis Reset'
  7 = 'Axis X'
  0 = 'Axis X '
  2 = 'Axis Y'
  3 = 'Axis Z'
  70 = 'Beckhoff Automation Turkey '
  26 = 'BW'
  112 = 'Cancel'
  55 = 'Cartesian Mode'
  110 = 'Checkbox'
  104 = 'Click for \nAuto Mode'
  105 = 'Click for \nManual Mode'
  21 = 'Deceleration'
  58 = 'DELTA ROBOT DEMOSET'
  93 = 'Drive Error'
  35 = 'Drive Reset'
  33 = 'DriveError'
  25 = 'Enable'
  12 = 'Error Id'
  43 = 'Finished'
  16 = 'Following Error'
  109 = 'G-Code List'
  29 = 'Home'
  24 = 'Home Pos'
  30 = 'Home Sensor'
  22 = 'Jerk'
  23 = 'Jog Velo'
  54 = 'Kin Execute'
  85 = 'KIN Group'
  56 = 'Kin Reset'
  1050 = 'Kinematic'
  53 = 'Kinematic Control'
  698 = 'Label'
  17 = 'Lag Distance'
  108 = 'Lag Distance[mm]'
  119 = 'Lag[mm]'
  80 = "M'"
  998 = 'M1 Pos Val'
  52 = 'M1_B'
  75 = 'M2'
  884 = 'M2 Pos Val'
  51 = 'M2_C'
  81 = 'M3'
  417 = 'M3 Pos Val'
  49 = 'M3_a'
  50 = 'M3_A'
  73 = 'Machine Coordinate System'
  71 = 'MAIN HMI '
  97 = 'Manual '
  101 = 'MANUAL MODE'
  92 = 'Manual Velocity'
  118 = 'MCS'
  95 = 'mm/s'
  87 = 'MODE'
  91 = 'MODE AUTOMATIC'
  89 = 'MODE MANUAL'
  90 = 'MODE OTOMATİK'
  31 = 'Move'
  38 = 'NCI Control'
  39 = 'NCI Enable'
  86 = 'NCI Group'
  45 = 'NCI Single'
  46 = 'NCI Single Mode'
  40 = 'NCI Start'
  47 = 'Next'
  36 = 'Open'
  57 = 'OpenFileDialog'
  88 = 'Otomatik'
  10 = 'Override'
  99 = 'Path'
  14 = 'Position'
  59 = 'POSITION M1'
  60 = 'Position M1'
  61 = 'Position M2'
  62 = 'Position M3'
  63 = 'Position X'
  64 = 'Position Y'
  65 = 'Position Z'
  106 = 'Position[mm]'
  67 = 'Power'
  102 = 'Press'
  103 = 'Press for \nAuto Mode'
  66 = 'R'
  34 = 'Reset'
  41 = 'Running'
  111 = 'Select'
  5 = 'Set. Position'
  48 = 'Single Mode'
  42 = 'Stopped'
  392 = 'Up'
  44 = 'Valve'
  15 = 'Velocity'
  107 = 'Velocity[mm/s]'
  98 = 'www.beckhoff.com.tr'
  82 = 'X'
  1066 = 'X Pos Val'
  750 = 'X+'
  420 = 'X-'
  83 = 'Y'
  120 = 'Y Pos Val'
  415 = 'Y+'
  1181 = 'Y-'
  84 = 'Z'
  1113 = 'Z Pos Val'
  809 = 'Z+'
  237 = 'Z-'
END_TEXTLIST

// ---- VISUs/Visualization_1.TcVIS
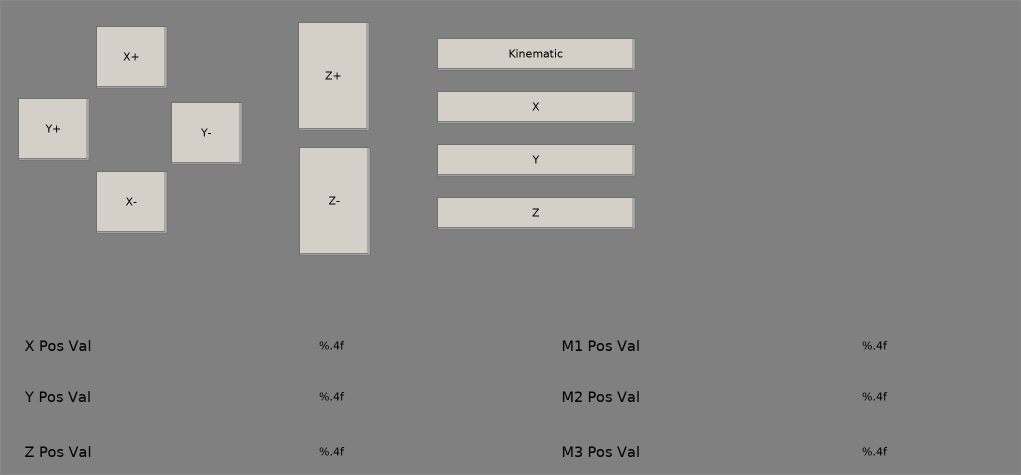
VISUALIZATION Visualization_1  // 1021x475
    Rectangle (187,334 289x24), "%.4f", text variable: GVL_Axis.AxisX.NcToPlc.ActPos
    Rectangle (187,385 289x24), "%.4f", text variable: GVL_Axis.AxisY.NcToPlc.ActPos
    Rectangle (187,440 289x24), "%.4f", text variable: GVL_Axis.AxisZ.NcToPlc.ActPos
    Label (10,325 96x42), "X Pos Val"
    Label (10,376 96x42), "Y Pos Val"
    Label (10,431 96x42), "Z Pos Val"
    Rectangle (730,334 289x24), "%.4f", text variable: GVL_Axis.AxisM1_B.NcToPlc.ActPos
    Rectangle (730,385 289x24), "%.4f", text variable: GVL_Axis.AxisM2_C.NcToPlc.ActPos
    Rectangle (730,440 289x24), "%.4f", text variable: GVL_Axis.AxisM3_A.NcToPlc.ActPos
    Label (553,325 96x42), "M1 Pos Val"
    Label (553,376 96x42), "M2 Pos Val"
    Label (553,431 96x42), "M3 Pos Val"
    Button (437,91 198x32), "X"
        OnMouseClick: toggle stAxisX.In.xMove
    Button (437,144 198x32), "Y"
        OnMouseClick: toggle stAxisY.In.xMove
    Button (437,197 198x32), "Z"
        OnMouseClick: toggle stAxisZ.In.xMove
    Button (437,38 198x32), "Kinematic"
        OnMouseClick: toggle PRG_Kinematic.bExecuteKinConfigGroup
    Button (96,26 71x62), "X+"
        tap POU_VisButton.xUp
    Button (96,171 71x62), "X-"
        tap POU_VisButton.xDown
    Button (171,102 71x62), "Y-"
        tap POU_VisButton.yDown
    Button (18,98 71x62), "Y+"
        tap POU_VisButton.yUp
    Button (298,22 71x108), "Z+"
        tap POU_VisButton.zuP
    Button (299,147 71x108), "Z-"
        tap POU_VisButton.zDown
END_VISUALIZATION

// ---- VISUs/Visualization_AxesInfo.TcVIS
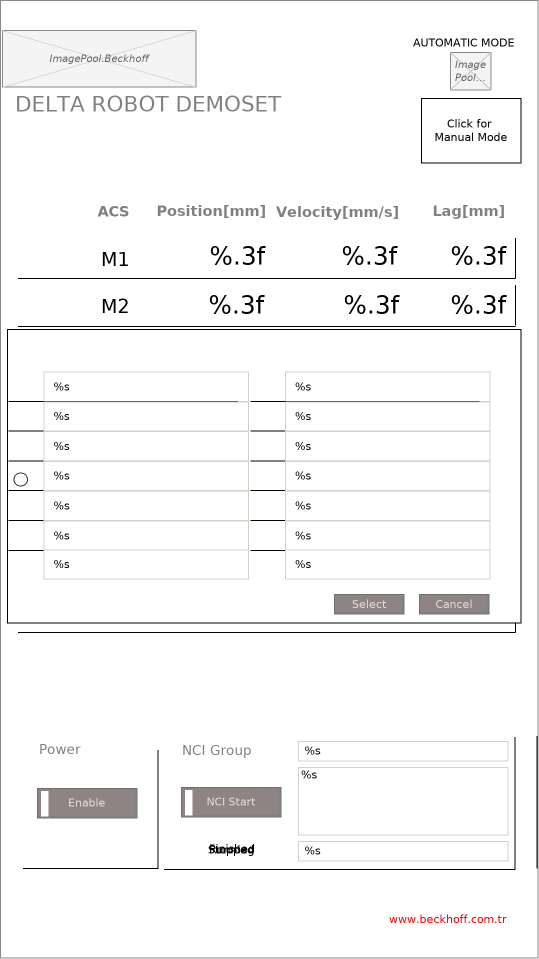
VISUALIZATION Visualization_AxesInfo  // 539x959, background image ImagePool.Background
    Label (35,229 155x61), "M1"
    Textfield (148,231 120x50), "%.3f", text variable: GVL_Axis.AxisM1_B.NcToPlc.ActPos
    Rectangle (39,248 7x22), invisible if: not stAxisM1_B.Out.xEnabled
    Rectangle (27,248 7x22), invisible if: not stAxisM1_B.Out.xAxisError
    Label (11,183 122x57), "ACS"
    Textfield (280,231 120x50), "%.3f", text variable: GVL_Axis.AxisM1_B.NcToPlc.ActVelo
    Image (2,30 194x57), image: ImagePool.Beckhoff
    Textfield (389,231 120x50), "%.3f", text variable: GVL_Axis.AxisM1_B.NcToPlc.PosDiff
    Line (18,278) (515,278)
    Line (515,238) (515,278)
    Label (38,276 155x61), "M2"
    Textfield (147,280 120x50), "%.3f", text variable: GVL_Axis.AxisM2_C.NcToPlc.ActPos
    Rectangle (39,295 7x22), invisible if: not stAxisM2_C.Out.xEnabled
    Rectangle (27,295 7x22), invisible if: not stAxisM2_C.Out.xAxisError
    Textfield (282,280 120x50), "%.3f", text variable: GVL_Axis.AxisM2_C.NcToPlc.ActVelo
    Textfield (389,280 120x50), "%.3f", text variable: GVL_Axis.AxisM2_C.NcToPlc.PosDiff
    Line (515,285) (515,325)
    Label (38,326 155x61), "M3"
    Textfield (147,330 120x50), "%.3f", text variable: GVL_Axis.AxisM3_A.NcToPlc.ActPos
    Rectangle (39,345 7x22), invisible if: not stAxisM3_A.Out.xEnabled
    Rectangle (27,345 7x22), invisible if: not stAxisM3_A.Out.xAxisError
    Textfield (282,330 120x50), "%.3f", text variable: GVL_Axis.AxisM3_A.NcToPlc.ActVelo
    Textfield (389,330 120x50), "%.3f", text variable: GVL_Axis.AxisM3_A.NcToPlc.PosDiff
    Line (18,376) (515,376)
    Line (515,335) (515,375)
    Line (18,326) (515,326)
    Label (11,447 122x57), "MCS"
    Label (8,493 120x50), "X"
    Textfield (126,488 140x50), "%.3f", text variable: GVL_Axis.AxisX.NcToPlc.ActPos
    Rectangle (39,505 7x22), invisible if: not stAxisX.Out.xEnabled
    Rectangle (27,505 7x22), invisible if: not stAxisX.Out.xAxisError
    Textfield (280,488 120x50), "%.3f", text variable: GVL_Axis.AxisX.NcToPlc.ActVelo
    Textfield (387,488 120x50), "%.3f", text variable: GVL_Axis.AxisX.NcToPlc.PosDiff
    Line (18,535) (515,535)
    Line (515,495) (515,535)
    Label (8,540 120x50), "Y"
    Textfield (126,537 140x50), "%.3f", text variable: GVL_Axis.AxisY.NcToPlc.ActPos
    Rectangle (39,552 7x22), invisible if: not stAxisY.Out.xEnabled
    Rectangle (27,552 6x22), invisible if: not stAxisY.Out.xAxisError
    Textfield (280,537 120x50), "%.3f", text variable: GVL_Axis.AxisY.NcToPlc.ActVelo
    Textfield (387,537 120x50), "%.3f", text variable: GVL_Axis.AxisY.NcToPlc.PosDiff
    Line (515,542) (515,582)
    Label (8,590 120x50), "Z"
    Textfield (126,587 140x50), "%.3f", text variable: GVL_Axis.AxisZ.NcToPlc.ActPos
    Rectangle (39,602 7x22), invisible if: not stAxisZ.Out.xEnabled
    Rectangle (27,602 7x22), invisible if: not stAxisZ.Out.xAxisError
    Textfield (280,587 120x50), "%.3f", text variable: GVL_Axis.AxisZ.NcToPlc.ActVelo
    Textfield (387,587 120x50), "%.3f", text variable: GVL_Axis.AxisZ.NcToPlc.PosDiff
    Line (18,632) (515,632)
    Line (515,592) (515,632)
    Line (17,583) (515,583)
    Textfield (298,767 210x68), "%s", text variable: PRG_NcControl.sNciLines
    Textfield (298,741 210x20), "%s", text variable: PRG_NcControl.sNciActualLine
    Label (189,834 86x30), "Finished", invisible if: NOT PRG_NcControl.bProgramFinished
    Label (188,835 86x30), "Stopped", invisible if: NOT PRG_NcControl.bProgramStopped
    Label (189,835 86x30), "Running", invisible if: NOT PRG_NcControl.bProgramRunning or PRG_NcControl.bProgramStopped
    Button (181,787 100x30), "NCI Start"
        toggle GVL_Process.bNciStartPLC
    Rectangle (185,790 7x25), invisible if: not PRG_NcControl.bNciStart
    Line (164,869) (515,869)
    Line (537,868) (537,736), invisible if: PRG_Process.bInvisible
    Label (147,722 140x57), "NCI Group"
    Textfield (298,841 210x20), "%s", text variable: PRG_Process.sFileNameVisu, input disabled if: PRG_NcControl.bProgramRunning
        toggle PRG_Process.bChangeFile
    Image (450,52 41x38), image: ImagePool.Mode_icon
        OnMouseMove: execute { GVL_Process.bMessageBubbleAuto := 1; }
        OnMouseClick: change screen: Visualization_AxesInfo_Manual
        OnMouseLeave: execute { GVL_Process.bMessageBubbleAuto := false; }
    Label (404,29 120x28), "AUTOMATIC MODE"
    Rectangle (421,98 100x65), "Click for Manual Mode", invisible if: not GVL_Process.bMessageBubbleAuto
    Frame (8,329 515x296), invisible if: not PRG_Process.bChangeFile
        shows Visualization_FileList()
    Label (12,77 308x54), "DELTA ROBOT DEMOSET"
    Label (149,186 120x50), "Position[mm]"
    Label (276,187 126x50), "Velocity[mm/s]"
    Label (388,186 120x50), "Lag[mm]"
    Button (37,788 100x30), "Enable"
        toggle GVL_Process.bAllAxesEnablePLC
    Rectangle (41,791 7x25), invisible if: not GVL_Process.bAllAxesEnable
    Line (23,868) (158,868)
    Line (158,868) (158,750)
    Label (25,721 70x57), "Power"
    Label (373,882 150x75), "www.beckhoff.com.tr"
    Line (515,869) (515,737)
END_VISUALIZATION

// ---- VISUs/Visualization_AxesInfo_Manual.TcVIS
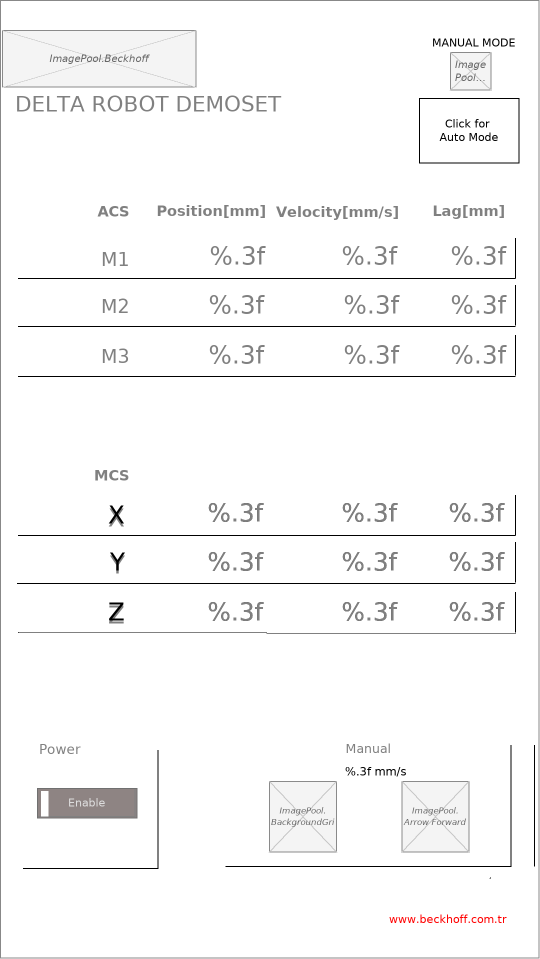
VISUALIZATION Visualization_AxesInfo_Manual  // 540x959, background image ImagePool.Background
    Textfield (8,590 120x50), "Z", invisible if: GVL_Process.bManualSelectZ
    Textfield (8,540 120x50), "Y", invisible if: GVL_Process.bManualSelectY
    Textfield (8,493 120x50), "X", invisible if: GVL_Process.bManualSelectX
    Textfield (8,537 120x50), "Y", invisible if: not GVL_Process.bManualSelectY
        p2073431371: GVL_Process.nSizeSelectY
    Frame (0,722 538x148)
        shows VisuAxisX_1()
        shows VisuAxisY_1()
        shows VisuAxisZ_1()
    Label (12,77 308x54), "DELTA ROBOT DEMOSET"
    Label (35,229 155x61), "M1"
    Textfield (148,231 120x50), "%.3f", text variable: GVL_Axis.AxisM1_B.NcToPlc.ActPos
    Rectangle (39,248 7x22), invisible if: not stAxisM1_B.Out.xEnabled
    Rectangle (27,248 7x22), invisible if: not stAxisM1_B.Out.xAxisError
    Label (11,183 122x57), "ACS"
    Label (149,186 120x50), "Position[mm]"
    Label (276,187 126x50), "Velocity[mm/s]"
    Textfield (280,231 120x50), "%.3f", text variable: GVL_Axis.AxisM1_B.NcToPlc.ActVelo
    Image (2,30 194x57), image: ImagePool.Beckhoff
    Label (388,186 120x50), "Lag[mm]"
    Textfield (389,231 120x50), "%.3f", text variable: GVL_Axis.AxisM1_B.NcToPlc.PosDiff
    Line (18,278) (515,278)
    Line (515,238) (515,278)
    Label (38,276 155x61), "M2"
    Textfield (147,280 120x50), "%.3f", text variable: GVL_Axis.AxisM2_C.NcToPlc.ActPos
    Rectangle (39,295 7x22), invisible if: not stAxisM2_C.Out.xEnabled
    Rectangle (27,295 7x22), invisible if: not stAxisM2_C.Out.xAxisError
    Textfield (282,280 120x50), "%.3f", text variable: GVL_Axis.AxisM2_C.NcToPlc.ActVelo
    Textfield (389,280 120x50), "%.3f", text variable: GVL_Axis.AxisM2_C.NcToPlc.PosDiff
    Line (515,285) (515,325)
    Label (38,326 155x61), "M3"
    Textfield (147,330 120x50), "%.3f", text variable: GVL_Axis.AxisM3_A.NcToPlc.ActPos
    Rectangle (39,345 7x22), invisible if: not stAxisM3_A.Out.xEnabled
    Rectangle (27,345 7x22), invisible if: not stAxisM3_A.Out.xAxisError
    Textfield (282,330 120x50), "%.3f", text variable: GVL_Axis.AxisM3_A.NcToPlc.ActVelo
    Textfield (389,330 120x50), "%.3f", text variable: GVL_Axis.AxisM3_A.NcToPlc.PosDiff
    Line (18,376) (515,376)
    Line (515,335) (515,375)
    Line (18,326) (515,326)
    Label (11,447 122x57), "MCS"
    Textfield (126,488 140x50), "%.3f", text variable: GVL_Axis.AxisX.NcToPlc.ActPos, invisible if: not GVL_Process.bManualSelectX
        p2073431371: GVL_Process.nSizeSelectX
    Rectangle (39,505 7x22), invisible if: not stAxisX.Out.xEnabled
    Rectangle (27,505 7x22), invisible if: not stAxisX.Out.xAxisError
    Textfield (280,488 120x50), "%.3f", text variable: GVL_Axis.AxisX.NcToPlc.ActVelo, invisible if: not GVL_Process.bManualSelectX
        p2073431371: GVL_Process.nSizeSelectX
    Textfield (387,488 120x50), "%.3f", text variable: GVL_Axis.AxisX.NcToPlc.PosDiff, invisible if: not GVL_Process.bManualSelectX
        p2073431371: GVL_Process.nSizeSelectX
    Line (18,535) (515,535), colour toggle: GVL_Process.bManualSelectX
    Line (515,495) (515,535), colour toggle: GVL_Process.bManualSelectX
    Textfield (126,537 140x50), "%.3f", text variable: GVL_Axis.AxisY.NcToPlc.ActPos, invisible if: not GVL_Process.bManualSelectY
        p2073431371: GVL_Process.nSizeSelectY
    Rectangle (39,552 7x22), invisible if: not stAxisY.Out.xEnabled
    Rectangle (27,552 7x22), invisible if: not stAxisY.Out.xAxisError
    Textfield (280,537 120x50), "%.3f", text variable: GVL_Axis.AxisY.NcToPlc.ActVelo, invisible if: not GVL_Process.bManualSelectY
        p2073431371: GVL_Process.nSizeSelectY
    Textfield (387,537 120x50), "%.3f", text variable: GVL_Axis.AxisY.NcToPlc.PosDiff, invisible if: not GVL_Process.bManualSelectY
        p2073431371: GVL_Process.nSizeSelectY
    Line (515,542) (515,582), colour toggle: GVL_Process.bManualSelectY
    Textfield (126,587 140x50), "%.3f", text variable: GVL_Axis.AxisZ.NcToPlc.ActPos, invisible if: not GVL_Process.bManualSelectZ
        p2073431371: GVL_Process.nSizeSelectZ
    Rectangle (39,602 7x22), invisible if: not stAxisZ.Out.xEnabled
    Rectangle (27,602 7x22), invisible if: not stAxisZ.Out.xAxisError
    Textfield (280,587 120x50), "%.3f", text variable: GVL_Axis.AxisZ.NcToPlc.ActVelo, invisible if: not GVL_Process.bManualSelectZ
        p2073431371: GVL_Process.nSizeSelectZ
    Textfield (387,587 120x50), "%.3f", text variable: GVL_Axis.AxisZ.NcToPlc.PosDiff, invisible if: not GVL_Process.bManualSelectZ
        p2073431371: GVL_Process.nSizeSelectZ
    Line (18,632) (515,633), colour toggle: GVL_Process.bManualSelectZ
    Line (515,592) (515,632), colour toggle: GVL_Process.bManualSelectZ
    Line (17,583) (515,583), colour toggle: GVL_Process.bManualSelectY
    Textfield (8,490 120x50), "X", invisible if: not GVL_Process.bManualSelectX
        p2073431371: GVL_Process.nSizeSelectX
    Textfield (8,587 120x50), "Z", invisible if: not GVL_Process.bManualSelectZ
        p2073431371: GVL_Process.nSizeSelectZ
    Textfield (126,537 140x50), "%.3f", text variable: GVL_Axis.AxisY.NcToPlc.ActPos, invisible if: GVL_Process.bManualSelectY
    Textfield (280,537 120x50), "%.3f", text variable: GVL_Axis.AxisY.NcToPlc.ActVelo, invisible if: GVL_Process.bManualSelectY
    Textfield (387,537 120x50), "%.3f", text variable: GVL_Axis.AxisY.NcToPlc.PosDiff, invisible if: GVL_Process.bManualSelectY
    Textfield (126,488 140x50), "%.3f", text variable: GVL_Axis.AxisX.NcToPlc.ActPos, invisible if: GVL_Process.bManualSelectX
    Textfield (280,488 120x50), "%.3f", text variable: GVL_Axis.AxisX.NcToPlc.ActVelo, invisible if: GVL_Process.bManualSelectX
    Textfield (387,488 120x50), "%.3f", text variable: GVL_Axis.AxisX.NcToPlc.PosDiff, invisible if: GVL_Process.bManualSelectX
    Textfield (126,587 140x50), "%.3f", text variable: GVL_Axis.AxisZ.NcToPlc.ActPos, invisible if: GVL_Process.bManualSelectZ
    Textfield (280,587 120x50), "%.3f", text variable: GVL_Axis.AxisZ.NcToPlc.ActVelo, invisible if: GVL_Process.bManualSelectZ
    Textfield (387,587 120x50), "%.3f", text variable: GVL_Axis.AxisZ.NcToPlc.PosDiff, invisible if: GVL_Process.bManualSelectZ
    Label (373,882 150x75), "www.beckhoff.com.tr"
    Group (23,721 136x148)
        Button (14,67 100x30), "Enable"
            toggle GVL_Process.bAllAxesEnable
        Rectangle (18,70 7x25), invisible if: not GVL_Process.bAllAxesEnable
        Line (0,147) (135,147)
        Line (135,147) (135,29)
        Label (2,0 70x57), "Power"
    InvisibleInput (8,485 510x51), input disabled if: GVL_Process.bManualSelectX
        toggle GVL_Process.bManualSelectX
        OnMouseClick: FrameSelectionChange Selection=SelectedFrame=4ba14cc2-2c84-48fd-8925-52c85ec640bd, GlobSel=AssignType=Directly, SelType=Locally
    InvisibleInput (8,585 510x51), input disabled if: GVL_Process.bManualSelectZ
        toggle GVL_Process.bManualSelectZ
        OnMouseClick: FrameSelectionChange Selection=SelectedFrame=4ba14cc2-2c84-48fd-8925-52c85ec640bd, Selection=2, GlobSel=AssignType=Directly, SelType=Locally
    InvisibleInput (8,535 510x51), input disabled if: GVL_Process.bManualSelectY
        toggle GVL_Process.bManualSelectY
        OnMouseClick: FrameSelectionChange Selection=SelectedFrame=4ba14cc2-2c84-48fd-8925-52c85ec640bd, Selection=1, GlobSel=AssignType=Directly, SelType=Locally
    Image (450,52 41x38), image: ImagePool.Mode_icon
        OnMouseMove: execute { GVL_Process.bMessageBubbleMan:=TRUE; }
        OnMouseClick: change screen: Visualization_AxesInfo
        OnMouseLeave: execute { GVL_Process.bMessageBubbleMan := FALSE; }
    Label (424,29 100x28), "MANUAL MODE"
    Rectangle (419,98 100x65), "Click for Auto Mode", invisible if: not GVL_Process.bMessageBubbleMan
    Rectangle (490,877 0x1)
END_VISUALIZATION
